// TIA Portal V16 export
// export: Created 2024-09-05T17:39:22.4466966Z, ExportSetting WithDefaults, DisplayName Totally Integrated Automation Portal, DisplayVersion V16 Update 6, DisplayName TIA Portal Version Control Interface, DisplayVersion V16 Update 2, DisplayName TIA Portal Openness, DisplayVersion V16 Update 6, DisplayName STEP 7 Professional, DisplayVersion V16 Update 6, DisplayName STEP 7 Safety, DisplayVersion V16, DisplayName WinCC Advanced, DisplayVersion V16 Update 6
DATA_BLOCK "ValueContinuityCheck_VH1_DB"   // DB44
VERSION : 0.1
// stored: AutoNumber true, DBAccessibleFromOPCUA true, InstanceOfName ValueContinuityCheck, InstanceOfType FB
"ValueContinuityCheck"
   // VAR_INPUT
   //    valueToCheck : Real;
   //    changeLimitForScan : Real;
   //    reset : Bool;
   // END_VAR
   // VAR_OUTPUT
   //    error : Bool;
   //    changeDuringError : Real;
   // END_VAR
   // VAR
   //    valueMemory : Real;
   //    biggestChange : Real;
   // END_VAR
BEGIN
END_DATA_BLOCK
